Fanuc KAREL source: kt00273.KL

-- PROVISIONAL review KL for V1013-1; original PC SHA256 14b60996786e3d7f7c763969c7cc129162e6aa2c509e77394cf5ddcda9299e17
-- Incomplete behavior may be omitted. Consult companion uncertainty JSON. Do not deploy.
PROGRAM KT00273
%NOLOCKGROUP
VAR
  OUT : BOOLEAN
-- UNRESOLVED_DECL H1 type=002017
-- UNRESOLVED_DECL Y2 type=002018
BEGIN
  -- UNRESOLVED_PC offsets 5-19; opcodes 2E,22,9D,33,B4
  -- UNRESOLVED_PC offsets 24-38; opcodes 2E,22,9D,33,B2
  -- UNRESOLVED_PC offsets 43-68; opcodes 22,9D,33,B3,22,9D,33,B1,57,23
  -- UNRESOLVED_PC offsets 73-77; opcodes 7F
END KT00273
